{attribute 'qualified_only'}
{attribute 'strict'}
TYPE eGridTripMode :
(
	Gridcode := 500,
	Default	:= 30,
	UPS		:= 10	
) UINT; //milliseconds
END_TYPE

(* stored: Version 1.1.0.1, ProductVersion 3.1.4026.18
   DUT eGridTripMode: Id {505d946e-68d4-456e-a198-ed5a25e79fb6} *)
